PROGRAM MAIN
VAR
END_VAR

END_PROGRAM

(* stored: Version 1.1.0.1
   POU MAIN: Id {22e0e3bd-d330-4fd0-8b10-abf6583da66e} *)
